{attribute 'qualified_only'}
TYPE ENUM_TwoTargets :
(
    Unknown := 0,
    OUT := 1,
    TARGET1 := 2,
    TARGET2 := 3
);
END_TYPE

(* stored: Version 1.1.0.1
   DUT ENUM_TwoTargets: Id {751a5e77-d869-49d5-873f-f68eb186a084} *)
